PROGRAM main
VAR
	BtnGreen AT %IX0.0 : bool;
	LEDGreen : bool;
	DECODER7SEG0 : Decoder7Seg;
END_VAR

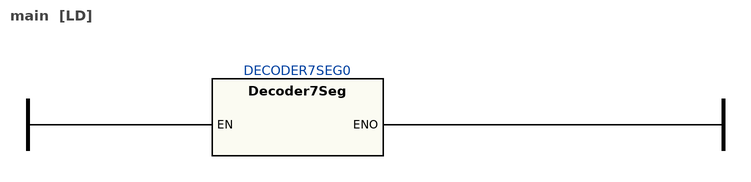
(* LD diagram, written out as Structured Text *)
DECODER7SEG0();
END_PROGRAM
